(* IEC 61131-3 sources: CodesysTest/export/Pro18.dev/Plc Logic/Application, 4 files *)

(* ---- PersistentVars.gvl.st ---- *)
(*#-#-#-#-#-#-#-#-#-#---Declaration---#-#-#-#-#-#-#-#-#-#-#-#-#*)

{attribute 'qualified_only'}
VAR_GLOBAL PERSISTENT RETAIN

	// Generated instance path of persistent variable
	Main_PRG.machineComponents.standardBagOpenFingersWithSensors.grabCounter.count: UDINT;
	// Generated instance path of persistent variable
	Main_PRG.machineComponents.standardBagOpenFingersWithSensors.releaseCounter.count: UDINT;
	// Generated instance path of persistent variable
	Main_PRG.machineComponents.standardBagOpenFingersWithSensors.missedCounter.count: UDINT;
	// Generated instance path of persistent variable
	HMI.data.pressureBarCycles.count: UDINT;
END_VAR

(* ---- FirstScan.pou.st ---- *)
(*#-#-#-#-#-#-#-#-#-#---Declaration---#-#-#-#-#-#-#-#-#-#-#-#-#*)

FUNCTION FirstScan : DWORD
VAR_IN_OUT
	EventPrm: CmpApp.EVTPARAM_CmpApp;
END_VAR
VAR
END_VAR(*#-#-#-#-#-#-#-#-#-#---Implementation---#-#-#-#-#-#-#-#-#-#-#-#-#*)

// Set first scan flag from StartDone system event
Globals.firstScan := TRUE;

(* ---- Devices.pou.st ---- *)
(*#-#-#-#-#-#-#-#-#-#---Declaration---#-#-#-#-#-#-#-#-#-#-#-#-#*)

PROGRAM Devices
VAR

END_VAR
VAR_IN_OUT

END_VAR

VAR_OUTPUT

	IOMaster : FB_MurrMaster(name := 'IO Master') := 	(ptrEIPInputs := ADR(IOEIPInputs),
														 ptrEIPOutputs := ADR(IOEIPOutputs));

	pressureBarSolenoidValve : FB_DoubleSolenoidOpenCenterActuator(name := 'Pressure Bar SV');
	sealBarSolenoidValve : FB_SingleSolenoidNormallyRetractedActuator(name := 'Seal Bar SV');
	HPA_LPA_SolenoidValve : FB_DoubleSolenoidClosedCenterActuator(name := 'HPA/LPA SV');
	loadPlateSolenoidValve : FB_DoubleSolenoidOpenCenterActuator(name := 'Load Plate SV');
	bagOpenFingersSolenoidValve : FB_DoubleSolenoidOpenCenterActuator(name := 'BOF SV');
	printHeadSolenoidValve : FB_SingleSolenoidNormallyRetractedActuator(name := 'Print Head SV');
	vacuumSolenoidValve : FB_VacuumGenerator(name := 'Vacuum SV');
	sealFlattenersVertAxisSolenoidValve : FB_DoubleSolenoidOpenCenterActuator(name := 'Seal Flattener Vert SV');
	loadShelfSolenoidValve : FB_DoubleSolenoidOpenCenterActuator(name := 'Load Shelf SV');
	blankSolenoidValve : FB_SolenoidValve(name := 'Blank SV');
	i : UINT;

	valveManifold : FB_SolenoidValveManifold(name := 'Valve Manifold') := (ptrEIPOutputs := ADR(Valve_Manifold_Outputs));

END_VAR
(*#-#-#-#-#-#-#-#-#-#---Implementation---#-#-#-#-#-#-#-#-#-#-#-#-#*)

// Valve manifold station selection
FOR i := 1 TO Globals.MAX_VALVE_MANIFOLD_STATIONS DO
	CASE HMI.data.stationValveSelection[i] OF

		ValveSelection.PressureBar : 						valveManifold.station[i] := pressureBarSolenoidValve;

		ValveSelection.SealBar : 							valveManifold.station[i] := sealBarSolenoidValve;

		ValveSelection.HPA_LPA : 							valveManifold.station[i] := HPA_LPA_SolenoidValve;

		ValveSelection.LoadPlate : 							valveManifold.station[i] := loadPlateSolenoidValve;

		ValveSelection.BagOpenFingers : 					valveManifold.station[i] := bagOpenFingersSolenoidValve;

		ValveSelection.PrintHead : 							valveManifold.station[i] := printHeadSolenoidValve;

		ValveSelection.Vacuum : 							valveManifold.station[i] := vacuumSolenoidValve;

		ValveSelection.SealFlattenersVerticalAxis : 		valveManifold.station[i] := sealFlattenersVertAxisSolenoidValve;

		ValveSelection.LoadShelf : 							valveManifold.station[i] := loadShelfSolenoidValve;

		ValveSelection.Blank : 								valveManifold.station[i] := blankSolenoidValve;

	ELSE
		valveManifold.station[i] := blankSolenoidValve;
	END_CASE
END_FOR

// Run all configured valves and then the manifold
pressureBarSolenoidValve();
sealBarSolenoidValve();
HPA_LPA_SolenoidValve();
loadPlateSolenoidValve();
bagOpenFingersSolenoidValve();
printHeadSolenoidValve();
vacuumSolenoidValve();
sealFlattenersVertAxisSolenoidValve();
loadShelfSolenoidValve();
blankSolenoidValve();
valveManifold();

IOMaster();

(* ---- Main_PRG.pou.st ---- *)
(*#-#-#-#-#-#-#-#-#-#---Declaration---#-#-#-#-#-#-#-#-#-#-#-#-#*)

PROGRAM Main_PRG
VAR

	firstScanDone : BOOL;
	UN00_Pro18Machine : FB_UN00_SharpMachine(name := 'UN00 - Sharp Pro-18');
	EM01_Pro18BaggerHead : EM01_BaggerHead(name := 'EM01 - Pro 18 Bagger Head');
	EM02_Pro18Discharge : EM02_Discharge(name := 'EM02 - Pro 18 Discharge');
	activeBaggerHead : REFERENCE TO EM01_BaggerHead;
	machineComponents : EM01_Bagger_Control_Modules();

	activeBagOpenFingers : IBagOpenFingers := machineComponents.standardBagOpenFingersWithSensors;
	activeSealFlatteners : ISealFlatteners;
	activePressureBar : IPressureBar;
	activeSealer : ISealer;
	activePrinter : IPrinter;
	activeBagDelivery : IBagDelivery;
	activeRetractingLoadPlate : IRetractingLoadPlate;
	activeExitConveyor : IExitConveyor;
	activeVacuumBagOpen : IVacuumBagOpen;

	powerUpPassthroughMotor : Sharp_Motion.MC_Power;
	powerUpMSFHorizMotor : Sharp_Motion.MC_Power;
	powerUpBagDeliveryMotor : Sharp_Motion.MC_Power;

END_VAR(*#-#-#-#-#-#-#-#-#-#---Implementation---#-#-#-#-#-#-#-#-#-#-#-#-#*)

{IF defined (IsSimulationMode)}
	HMI.data.simulateAllIO := TRUE;
{END_IF}

Devices();
machineComponents();

powerUpPassthroughMotor(Enable := TRUE, Axis := machineComponents.passthroughMotor);
powerUpPassthroughMotor.DriveStart := TRUE;
powerUpPassthroughMotor.RegulatorOn := TRUE;

powerUpMSFHorizMotor(Enable := TRUE, Axis := machineComponents.msfHorizontalMotor);
powerUpMSFHorizMotor.DriveStart := TRUE;
powerUpMSFHorizMotor.RegulatorOn := TRUE;

powerUpBagDeliveryMotor(Enable := TRUE, Axis := machineComponents.bagDeliveryFrontMotor);
powerUpBagDeliveryMotor.DriveStart := TRUE;
powerUpBagDeliveryMotor.RegulatorOn := TRUE;

CASE HMI.data.bofSelection OF
	BagOpenFingersSelection.NotInstalled:
															activeBagOpenFingers := machineComponents.standardBagOpenFingersWithSensors;
															activeBagOpenFingers.OptionInstalled := FALSE;

	BagOpenFingersSelection.PneumaticWithBagOpenSensors: 	activeBagOpenFingers := machineComponents.standardBagOpenFingersWithSensors;
															activeBagOpenFingers.OptionInstalled := TRUE;
															activeBagOpenFingers.OptionEnabled := HMI.data.bofEnable;
END_CASE

CASE HMI.data.sealFlattenersSelection OF
	SealFlattenerSelection.NotInstalled:					activeSealFlatteners := machineComponents.motorizedSealFlatteners;
															activeSealFlatteners.OptionInstalled := FALSE;

	SealFlattenerSelection.MotorizedSealFlatteners:			activeSealFlatteners := machineComponents.motorizedSealFlatteners;
															activeSealFlatteners.OptionInstalled := TRUE;
															activeSealFlatteners.OptionEnabled := HMI.data.sealFlattenersEnable;
END_CASE

CASE HMI.data.printerSelection OF
	LabelPrinterSelection.NotInstalled:						activePrinter := machineComponents.labelPrinter;
															activePrinter.OptionInstalled := FALSE;

	LabelPrinterSelection.ZebraPrinter:						activePrinter := machineComponents.labelPrinter;
															activePrinter.OptionInstalled := TRUE;
															activePrinter.OptionEnabled := HMI.data.printerEnable;
END_CASE

EM01_Pro18BaggerHead(
	bagOpenFingers:= activeBagOpenFingers,
	sealFlatteners:= activeSealFlatteners,
	sealer:= machineComponents.standardSealBar,
	pressureBar:= machineComponents.pneumaticPressureBar,
	printer:= activePrinter,
	bagDelivery:= machineComponents.bagDelivery,
	vacuumBagOpen:= machineComponents.vacuumCups,
	bagOpenAssistEnabled:= HMI.data.bagOpenAssistEnable,
	bagOpenSensorEnabled:= HMI.data.bagOpenSensorEnable,
	separateBeforeSealEnabled:= HMI.data.separateBeforeSeal,
	bagOpenRetrySetting:= HMI.data.bagOpenRetrySetting,
	vacuumDwell := TO_TIME(HMI.data.vacuumDwell * 1000),
	baggerCycleActive=> ,
	bagOpenRetryCount=> HMI.data.bagOpenRetryCount);

activeBaggerHead REF= EM01_Pro18BaggerHead;
UN00_Pro18Machine(
	faultActive := HMI.data.faultActive,
	baggerHead := activeBaggerHead,
	discharge := EM02_Pro18Discharge);

Globals.SystemLog();

IF NOT firstScanDone THEN
	GlobalObjects.CollectionOfInitialzable.InitializeAll();
	GlobalObjects.CollectionOfLoggable.RegisterAll(internalLogger := Globals.SystemLog);
	GlobalObjects.CollectionOfFaults.FaultUpdateForHMI();
	firstScanDone := TRUE;
END_IF

HMI.data.faultActive := GlobalObjects.CollectionOfActiveFaults.faultActive;
IF HMI.data.ackAllFaults THEN
	GlobalObjects.CollectionOfActiveFaults.AckAll();
	HMI.data.ackAllFaults := FALSE;
END_IF

IF HMI.data.initiateCycle THEN
	IF UN00_Pro18Machine.currentState = PACK_ML.State.Execute THEN
		activeBaggerHead.StartCycle();
	END_IF
	HMI.data.initiateCycle := FALSE;
END_IF

IF firstScanDone THEN
	GlobalObjects.CollectionOfExecutable.ExecuteAll();
END_IF
